// TIA Portal V16 export
// export: Created 2024-12-03T15:41:43.3980745Z, ExportSetting WithDefaults, DisplayName Totally Integrated Automation Portal, DisplayVersion V16 Update 6, DisplayName TIA Portal Version Control Interface, DisplayVersion V16 Update 2, DisplayName TIA Portal Openness, DisplayVersion V16 Update 6, DisplayName TIA Portal Teamcenter Gateway, DisplayVersion V16, DisplayName SINAMICS Startdrive Advanced, DisplayVersion V16 Update 5, DisplayName SINAMICS Startdrive G130, G150, S120, S150, SINAMICS MV, S210, DisplayVersion V16 Update 5, DisplayName SINAMICS Startdrive G110M, G120, G120C, G120D, G120P, G115D, DisplayVersion V16 Update 5, DisplayName STEP 7 Professional, DisplayVersion V16 Update 6, DisplayName STEP 7 Safety, DisplayVersion V16, DisplayName WinCC Advanced / Unified PC, DisplayVersion V16 Update 6
FUNCTION_BLOCK "TrafficController_INTERSECT_RECEIVE_FB"   // FB54, SCL
{ S7_Optimized_Access := 'TRUE' }
VERSION : 0.1
// intersection receives from one section and can sent to other 3 sections
// stored: AutoNumber true, IsIECCheckEnabled false, IsRetainMemResEnabled false, MemoryReserve 100, SetENOAutomatically false, UDAEnableTagReadback false
   VAR_INPUT
      I_IntersectionConveyor : "Conveyor_UDT";
      I_Option_1_Settings { ExternalAccessible := 'False'; ExternalVisible := 'False'; ExternalWritable := 'False'} : "Intersection";   // Intersection settings for option 1 (no split executed)
      I_Option_2_Settings { ExternalAccessible := 'False'; ExternalVisible := 'False'; ExternalWritable := 'False'} : "Intersection";   // Intersection settings for option 2 (split executed)
   END_VAR
   VAR_IN_OUT
      IO_IntersectionSettings : "Intersection";
      IO_SendingConveyor_1 : "Conveyor_UDT";   // The main conveyor on the intersection
      IO_SendingConveyor_2 : "Conveyor_UDT";
   END_VAR
   VAR
      unlockDelay : TON_TIME;
      empty { S7_SetPoint := 'True'} : "SmartBool";
      LOCK : Bool;
      option : Int;
      OptionsSaved : Bool;
      conv1_wait : DInt;
      conv2_wait : DInt;
      cycle { S7_SetPoint := 'True'} : "ScanTimer_FB";
   END_VAR
   VAR_TEMP
      T_Condition : Bool;
   END_VAR
BEGIN
   #IO_SendingConveyor_1.Cmd.Accumulate.Acc_TC_1 := TRUE;
   #IO_SendingConveyor_2.Cmd.Accumulate.Acc_TC_1 := TRUE;

   REGION FLOW CONTROL

       REGION CALCULATE WAIT TIMES
           #cycle();

           IF #IO_SendingConveyor_1.Status.RequestForSending THEN
               #conv1_wait += #cycle.O_ScanTime;
           ELSE
               #conv1_wait := 0;
           END_IF;

           IF #IO_SendingConveyor_2.Status.RequestForSending THEN
               #conv2_wait += #cycle.O_ScanTime;
           ELSE
               #conv2_wait := 0;
           END_IF;

       END_REGION

       //#option := 0;

       IF #conv1_wait > 0 AND #conv1_wait >= #conv2_wait AND NOT #LOCK THEN
           #option := 1;
           #LOCK := 1;
       END_IF;

       IF #conv2_wait > 0 AND #conv2_wait > #conv1_wait AND NOT #LOCK THEN
           #option := 2;
           #LOCK := 1;
       END_IF;

   END_REGION

   REGION CHECK TO TRANSFER SETTINGS

       IF (#IO_SendingConveyor_1.Status.RequestForSending OR #IO_SendingConveyor_2.Status.RequestForSending)
           AND #I_IntersectionConveyor.Status.Empty THEN

           CASE #option OF
               1:
                   #IO_IntersectionSettings := #I_Option_1_Settings;
               2:
                   #IO_IntersectionSettings := #I_Option_2_Settings;
           END_CASE;


       END_IF;

   END_REGION

   REGION TURN OFF ACCUMULATION OF SENDING CONV

       IF (#IO_SendingConveyor_1.Status.RequestForSending OR #IO_SendingConveyor_2.Status.RequestForSending)
           AND #I_IntersectionConveyor.Status.Empty THEN

           IF #option = 1 THEN
               #IO_SendingConveyor_1.Cmd.Accumulate.Acc_TC_1 := FALSE;
           END_IF;

           IF #option = 2 THEN
               #IO_SendingConveyor_2.Cmd.Accumulate.Acc_TC_1 := FALSE;
           END_IF;

       END_IF;

   END_REGION

   REGION UNLOCK

       #empty(I_Sensor := #I_IntersectionConveyor.Status.Empty);

       #T_Condition :=
       #I_IntersectionConveyor.Status.Empty AND
       NOT #IO_SendingConveyor_1.Cmd.RunAuto AND
       NOT #IO_SendingConveyor_2.Cmd.RunAuto AND
       #LOCK;

       #unlockDelay(IN := #T_Condition,
                    PT := t#3s);


       IF #empty.O_data.LE OR #unlockDelay.Q THEN
           #LOCK := 0;
       END_IF;

   END_REGION
END_FUNCTION_BLOCK
